SYSTEM StructRenameTest
  (* Version 1.0, 2026-05-31, Dimitrios Kalligaridis *)
  APPLICATION App
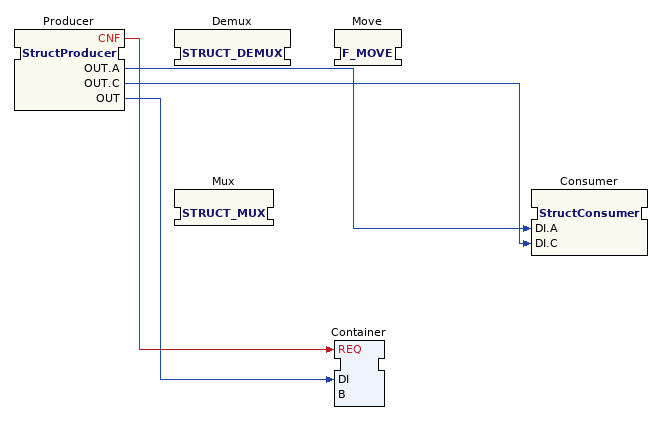
    FBS
      Producer : StructProducer(OUT.A :=  {SET_ATTRIBUTE(TestAttribute, 42)});
      Demux : STRUCT_DEMUX; {SET_ATTRIBUTE(StructuredType, mypackage::InnerStruct)} {SET_ATTRIBUTE(VisibleChildren, A,C)}
      Mux : STRUCT_MUX; {SET_ATTRIBUTE(StructuredType, mypackage::InnerStruct)}
      Move : F_MOVE; {SET_ATTRIBUTE(DataType, mypackage::InnerStruct)}
      Consumer : StructConsumer;
    END_FBS
    SUBAPPLICATION Container
      EVENT_INPUT
        REQ;
      END_EVENT
      VAR_INPUT
        DI : mypackage::InnerStruct;
        B : BOOL;
      END_VAR
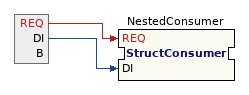
      FBS
        NestedConsumer : StructConsumer;
      END_FBS
      EVENT_CONNECTIONS
        REQ TO NestedConsumer.REQ;
      END_CONNECTIONS
      DATA_CONNECTIONS
        DI TO NestedConsumer.DI;
      END_CONNECTIONS
    END_SUBAPPLICATION
    EVENT_CONNECTIONS
      Producer.CNF TO Container.REQ;
    END_CONNECTIONS
    DATA_CONNECTIONS
      Producer.OUT.A TO Consumer.DI.A;
      Producer.OUT.C TO Consumer.DI.C;
      Producer.OUT TO Container.DI;
    END_CONNECTIONS
  END_APPLICATION
END_SYSTEM
